FUNCTION_BLOCK IOManager
  (* Standard: 61499-2 *)
  (* Version 0.1, 2016-00-28, hpea485, UOA *)
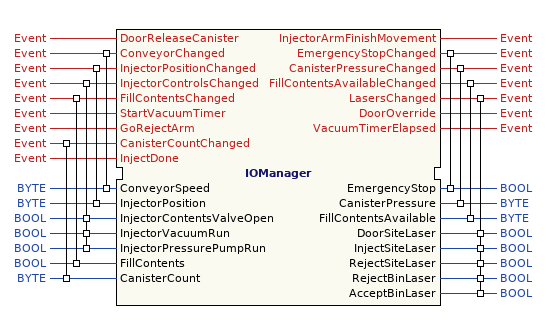
  EVENT_INPUT
    DoorReleaseCanister;
    ConveyorChanged WITH ConveyorSpeed;
    InjectorPositionChanged WITH InjectorPosition;
    InjectorControlsChanged WITH InjectorContentsValveOpen, InjectorVacuumRun, InjectorPressurePumpRun;
    FillContentsChanged WITH FillContents;
    StartVacuumTimer;
    GoRejectArm;
    CanisterCountChanged WITH CanisterCount;
    InjectDone;
  END_EVENT
  EVENT_OUTPUT
    InjectorArmFinishMovement;
    EmergencyStopChanged WITH EmergencyStop;
    CanisterPressureChanged WITH CanisterPressure;
    FillContentsAvailableChanged WITH FillContentsAvailable;
    LasersChanged WITH DoorSiteLaser, InjectSiteLaser, RejectSiteLaser, RejectBinLaser, AcceptBinLaser;
    DoorOverride;
    VacuumTimerElapsed;
  END_EVENT
  VAR_INPUT
    ConveyorSpeed : BYTE;
    InjectorPosition : BYTE;
    InjectorContentsValveOpen : BOOL;
    InjectorVacuumRun : BOOL;
    InjectorPressurePumpRun : BOOL;
    FillContents : BOOL;
    CanisterCount : BYTE;
  END_VAR
  VAR_OUTPUT
    EmergencyStop : BOOL;
    CanisterPressure : BYTE;
    FillContentsAvailable : BYTE;
    DoorSiteLaser : BOOL;
    InjectSiteLaser : BOOL;
    RejectSiteLaser : BOOL;
    RejectBinLaser : BOOL;
    AcceptBinLaser : BOOL;
  END_VAR
  VAR
    EmergencyStopped : INT := 1;
    BottlePositions : ARRAY [0..3] OF INT := [0,0,0,0];
    BottlesActive : ARRAY [0..3] OF BOOL := [0,0,0,0];
    NextBottle : INT := 0;
    InternalConveyorSpeed : INT := 0;
  END_VAR
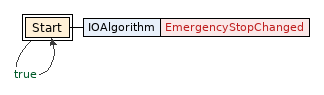
  EC_STATES
    Start : IOAlgorithm -> EmergencyStopChanged;
  END_STATES
  EC_TRANSITIONS
    Start TO Start := true;
  END_TRANSITIONS
  ALGORITHM IOAlgorithm IN C:
#define NUM_BOTTLES 4

int i;

//reset all the things
me->EmergencyStop = 0;
me->CanisterPressure = 255;
me->FillContentsAvailable = 255;
me->DoorSiteLaser = 0;
me->InjectSiteLaser = 0;
me->RejectSiteLaser = 0;
me->RejectBinLaser = 0;
me->AcceptBinLaser = 0;


//printf("=====new tick\n");

//continue progress
if(me->ConveyorSpeed) {
	for(i = 0; i < 4; i++) {
		if(me->BottlesActive[i]) {
			me->BottlePositions[i] += me->InternalConveyorSpeed;
			printf("IO: Canister %i moves to %i\n", i, me->BottlePositions[i]);

			if(me->BottlePositions[i] == 5) {
				printf("IO: Canister %i at 5, triggering InjectSiteLaser\n", i);
				me->outputEvents.event.LasersChanged = 1;
				me->InjectSiteLaser = 1;
			} else if(me->BottlePositions[i] == 10) {
				printf("IO: Canister %i at 10, triggering RejectSiteLaser\n", i);
				me->outputEvents.event.LasersChanged = 1;
				me->RejectSiteLaser = 1;
			} else if(me->BottlePositions[i] == 20) {
				printf("IO: Canister %i at 20, falls off conveyor, triggering AcceptBinLaser\n", i);
				me->outputEvents.event.LasersChanged = 1;
				me->AcceptBinLaser = 1;
				me->BottlesActive[i] = 0;
				me->BottlePositions[i] = 0;
			}

			if(me->inputEvents.event.GoRejectArm && (me->BottlePositions[i] == 10 || me->BottlePositions[i] == 11 || me->BottlePositions[i] == 12)) {
				printf("IO: Go Reject Arm. Canister %i knocked from conveyor.\n", i);
				//progress = 0;
				me->outputEvents.event.LasersChanged = 1;
				me->RejectBinLaser = 1;
				me->BottlesActive[i] = 0;
				me->BottlePositions[i] = 0;
			}
		}
	}
}

//if(canisterProgress == 25) {
//	printf("Progress at 25, halting\n");
//	while(1);
//}

if(me->inputEvents.event.InjectDone) {
	printf("IO: Inject done\n");
}



if(me->EmergencyStopped == 1) {
	printf("IO: Releasing emergency stop\n");
	me->outputEvents.event.EmergencyStopChanged = 1;
	me->EmergencyStop = 0;
	me->EmergencyStopped++;
} else {

	if(me->inputEvents.event.DoorReleaseCanister) {
		printf("IO: Door released. Adding canister %i\n", me->NextBottle);

		me->outputEvents.event.LasersChanged = 1;
		me->DoorSiteLaser = 1;

		me->BottlesActive[me->NextBottle] = 1;

		me->NextBottle++;
		me->NextBottle = me->NextBottle % 4;

	}
	if(me->inputEvents.event.InjectorPositionChanged) {
		printf("IO: Injector position changed. Setting move finished.\n");
		me->outputEvents.event.InjectorArmFinishMovement = 1;
	}

	if(me->inputEvents.event.ConveyorChanged) {
		me->InternalConveyorSpeed = me->ConveyorSpeed;
		printf("IO: Setting conveyor movement to %i\n", me->InternalConveyorSpeed);
	}



	if(me->inputEvents.event.InjectorControlsChanged) {
		printf("IO: Injector controls changed. Now they are Vac: %1i Val: %1i Pmp: %1i\n", me->InjectorVacuumRun, me->InjectorContentsValveOpen, me->InjectorPressurePumpRun);
		if(me->InjectorVacuumRun) {
			printf("IO: Due to vacuum, changing canister pressure to 5.\n");
			me->CanisterPressure = 5;
			me->outputEvents.event.CanisterPressureChanged = 1;
		}
		if(me->InjectorContentsValveOpen) {
			printf("IO: Contents valve now open. Pressure changes slightly, sucking in contents.\n");
			me->CanisterPressure = 20;
			me->outputEvents.event.CanisterPressureChanged = 1;
		}
		if(me->InjectorPressurePumpRun) {
			printf("IO: Due to pressure pump, changing canister pressure to 250.\n");
			me->CanisterPressure = 250;
			me->outputEvents.event.CanisterPressureChanged = 1;
		}
	}

	if(me->inputEvents.event.FillContentsChanged) {
		printf("IO: Fill contents changed.\n");
	}

	if(me->inputEvents.event.StartVacuumTimer) {
		printf("IO: Start vacuum timer.\n");//Elapsing timer.\n");
		//me->outputEvents.event.VacuumTimerElapsed = 1;
	}



	if(me->inputEvents.event.CanisterCountChanged) {
		printf("IO: Canister count changed. New value: %i\n", me->CanisterCount);
	}


}
  END_ALGORITHM
END_FUNCTION_BLOCK
